// TIA Portal V20 export
VAR_GLOBAL   // PLC tag table "Profinet_Comunication"
   Tag_1 AT %IB532 : Byte;
   Tag_2 AT %IB534 : Byte;
   Tag_3 AT %ID518 : DWord;
END_VAR
